TYPE JointState :
STRUCT
	Position : Joints;
	Velocity : Joints;
	Current  : Joints;
END_STRUCT
END_TYPE

(* stored: Version 1.1.0.1, ProductVersion 3.1.0.36
   DUT JointState: Id {e43395f1-3fb0-4070-a889-ed79cf1f4551} *)
